(* Schneider Machine Expert - Basic project memory floats gt, file version 2.0.0.0 *)
(* ProjectInformations: Name=New project *)

HARDWARE
  Cpu 0: TM221M16R/G
  EthernetConfiguration: NetworkName=M221, IpAllocationMode=FixedAddress, IpAddress=0.0.0.0, SubnetMask=0.0.0.0
  SerialLineConfiguration: Baud=Baud19200, Parity=ParityEven, DataBits=DataBits8, StopBits=StopBits1, PhysicalMedium=PhysicalMediumRs485, TransmissionMode=TransmissionModeModbusRtu, SlaveId=1, Addressing=SlaveAddressing
  MastTask: UsePeriodScanMode=false, PeriodScan=100
  FastTask: Period=255
  CpuBehavior: StartingMode=StartAsPreviousState, AutoSaveRamOnEeprom=true, WatchdogPeriod=250

SYMBOLS  (address, symbol, comment, settings)

POU New POU
  (* SectionNumber=1 *)

// Rung 0
  LD %I0.0
  OPER [ %MF2 := 1.0 ]
  ST %Q0.0
  // as ST:
  //   IF %I0.0 THEN %MF2 := 1.0; END_IF;
  //   %Q0.0 := %I0.0;

// Rung 1
  LD %I0.0
  AND [ %MF1 <= %MF2 ]
  ST %Q0.0
  // as ST:
  //   %Q0.0 := %I0.0 AND %MF1 <= %MF2;

// Rung 2
  LD %I0.0
  AND [ %MF1 > %MF2 ]
  ST %Q0.0
  // as ST:
  //   %Q0.0 := %I0.0 AND %MF1 > %MF2;

// Rung 3
  LD %I0.0
  AND [ %MF1 >= %MF2 ]
  ST %Q0.0
  // as ST:
  //   %Q0.0 := %I0.0 AND %MF1 >= %MF2;

// Rung 4
  LD %I0.0
  AND [ %MF1 <> %MF2 ]
  ST %Q0.0
  // as ST:
  //   %Q0.0 := %I0.0 AND %MF1 <> %MF2;

// Rung 5
  LD %I0.0
  AND [ %MF1 = %MF2 ]
  ST %Q0.0
  // as ST:
  //   %Q0.0 := %I0.0 AND %MF1 = %MF2;

// Rung 6
  LD %I0.0
  AND [ %MF1 = %MF1 + %MF2 ]
  ST %Q0.0
  // as ST:
  //   %Q0.0 := %I0.0 AND %MF1 = %MF1 + %MF2;

// Rung 7
  LD %I0.0
  AND [ %MF1 = %MF1 - %MF2 ]
  ST %Q0.0
  // as ST:
  //   %Q0.0 := %I0.0 AND %MF1 = %MF1 - %MF2;

// Rung 8
  LD %I0.0
  AND [ %MF1 = %MF1 * %MF2 ]
  ST %Q0.0
  // as ST:
  //   %Q0.0 := %I0.0 AND %MF1 = %MF1 * %MF2;

// Rung 9
  LD %I0.0
  AND [ %MF1 = %MF1 / %MF2 ]
  ST %Q0.0
  // as ST:
  //   %Q0.0 := %I0.0 AND %MF1 = %MF1 / %MF2;

// Rung 10
  LD %I0.0
  AND [ %MF1 = 1.0 + %MF2 ]
  ST %Q0.0
  // as ST:
  //   %Q0.0 := %I0.0 AND %MF1 = 1.0 + %MF2;

// Rung 11
  LD %I0.0
  AND [ %MF1 = 1.0 - %MF2 ]
  ST %Q0.0
  // as ST:
  //   %Q0.0 := %I0.0 AND %MF1 = 1.0 - %MF2;

// Rung 12
  LD %I0.0
  AND [ %MF1 = 1.0 * %MF2 ]
  ST %Q0.0
  // as ST:
  //   %Q0.0 := %I0.0 AND %MF1 = 1.0 * %MF2;

// Rung 13
  LD %I0.0
  AND [ %MF1 = 1.0 / %MF2 ]
  ST %Q0.0
  // as ST:
  //   %Q0.0 := %I0.0 AND %MF1 = 1.0 / %MF2;

// Rung 14
  LD %I0.0
  OPER [ %MF1 := 1.0 / %MF2 ]
  ST %Q0.0
  // as ST:
  //   IF %I0.0 THEN %MF1 := 1.0 / %MF2; END_IF;
  //   %Q0.0 := %I0.0;

// Rung 15
  LD %I0.0
  OPER [ %MF1 := 2.0 + %MF2 ]
  ST %Q0.0
  // as ST:
  //   IF %I0.0 THEN %MF1 := 2.0 + %MF2; END_IF;
  //   %Q0.0 := %I0.0;

// Rung 16
  LD %I0.0
  AND [ %MF1 = ( 2.0 * 3.0 ) * ( %MF2 + %MF3 ) ]
  ST %Q0.0
  // as ST:
  //   %Q0.0 := %I0.0 AND %MF1 = ( 2.0 * 3.0 ) * ( %MF2 + %MF3 );

// Rung 17
  LD %I0.0
  AND [ %MF1 = 2.0 + 3.0 ]
  ST %Q0.0
  // as ST:
  //   %Q0.0 := %I0.0 AND %MF1 = 2.0 + 3.0;

// Rung 18
  LD %I0.0
  AND [ %MF1 = 2.0 - 3.0 ]
  ST %Q0.0
  // as ST:
  //   %Q0.0 := %I0.0 AND %MF1 = 2.0 - 3.0;

// Rung 19
  LD %I0.0
  AND [ %MF1 = 2.0 * 3.0 ]
  ST %Q0.0
  // as ST:
  //   %Q0.0 := %I0.0 AND %MF1 = 2.0 * 3.0;

// Rung 20
  LD %I0.0
  AND [ %MF1 = 2.0 / 3.0 ]
  ST %Q0.0
  // as ST:
  //   %Q0.0 := %I0.0 AND %MF1 = 2.0 / 3.0;

// Rung 21
  LD %I0.0
  AND [ %MF1 < 1.0 ]
  ST %Q0.0
  // as ST:
  //   %Q0.0 := %I0.0 AND %MF1 < 1.0;

// Rung 22
  LD %I0.0
  AND [ %MF1 <= 1.0 ]
  ST %Q0.0
  // as ST:
  //   %Q0.0 := %I0.0 AND %MF1 <= 1.0;

// Rung 23
  LD %I0.0
  AND [ %MF1 > 1.0 ]
  ST %Q0.0
  // as ST:
  //   %Q0.0 := %I0.0 AND %MF1 > 1.0;

// Rung 24
  LD %I0.0
  AND [ %MF1 >= 1.0 ]
  ST %Q0.0
  // as ST:
  //   %Q0.0 := %I0.0 AND %MF1 >= 1.0;

// Rung 25
  LD %I0.0
  AND [ %MF1 = 1.0 ]
  ST %Q0.0
  // as ST:
  //   %Q0.0 := %I0.0 AND %MF1 = 1.0;

// Rung 26
  LD %I0.0
  AND [ %MF1 <> 1.0 ]
  ST %Q0.0
  // as ST:
  //   %Q0.0 := %I0.0 AND %MF1 <> 1.0;
